DATA_BLOCK "dbArchiveSlotEom"
{ S7_Optimized_Access := 'TRUE' }
VERSION : 0.8
NON_RETAIN
"fbArchiveSlotEom"

BEGIN

END_DATA_BLOCK

